KUKA KRL program: Milling_2_2.src

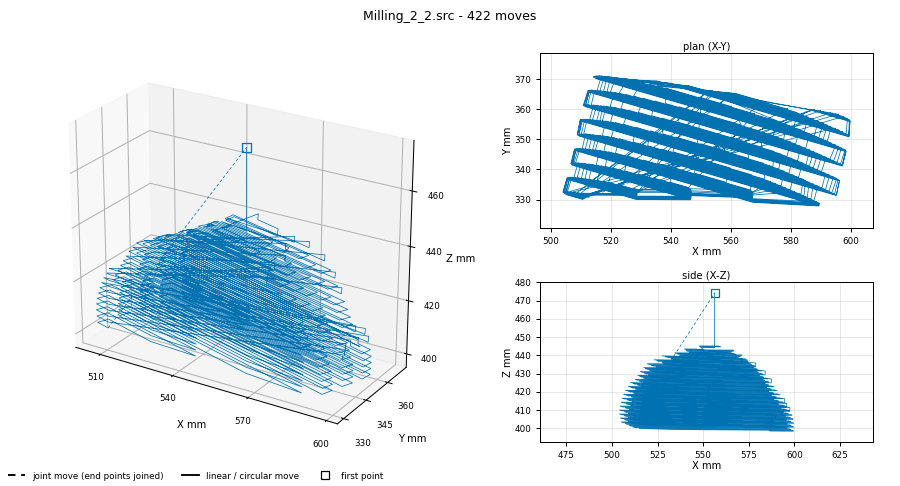
[picture p0: tool path of Milling_2_2.src, 422 of 424 moves have a stored position in this frame; points joined in program order, loops and branches not executed]
&ACCESS RVP
&REL 1
&PARAM TEMPLATE = C:\KRC\Roboter\Template\vorgabe
&PARAM EDITMASK = *
DEF Milling_2_2 ( )


;FOLD INI
;FOLD BASISTECH INI
GLOBAL INTERRUPT DECL 3 WHEN $STOPMESS==TRUE DO IR_STOPM ( )
INTERRUPT ON 3
BAS (#INITMOV,0 )
;ENDFOLD (BASISTECH INI)
;ENDFOLD (INI)

;FOLD STARTPOSITION - BASE IS 0, TOOL IS 5, SPEED IS 15%, POSITION IS A1 5,A2 -90,A3 100,A4 5,A5 -10,A6 -5,E1 0,E2 0,E3 0,E4 0
$BWDSTART = FALSE
PDAT_ACT = {VEL 15,ACC 100,APO_DIST 50}
FDAT_ACT = {TOOL_NO 5,BASE_NO 0,IPO_FRAME #BASE}
BAS (#PTP_PARAMS,15)
PTP  {A1 5,A2 -90,A3 100,A4 5,A5 -10,A6 -5,E1 0,E2 0,E3 0,E4 0}
;ENDFOLD

;FOLD LIN SPEED IS 0.1 m/sec, INTERPOLATION SETTINGS IN FOLD
$VEL.CP=0.1
$ADVANCE=3
;ENDFOLD

BAS(#VEL_PTP,2)
PTP {X 556.311, Y 346.712, Z 474.273, A -110.612, B 84.801, C -94.37, E1 0, E2 0, E3 0, E4 0, S 'B010'}
$VEL.CP=0.012
LIN {X 556.311, Y 346.712, Z 444.273, A -110.612, B 84.801, C -94.37, E1 0, E2 0, E3 0, E4 0}
LIN {X 549.895, Y 348.583, Z 444.319, A -110.612, B 84.801, C -94.37, E1 0, E2 0, E3 0, E4 0}
LIN {X 548.876, Y 343.693, Z 444.768, A -110.612, B 84.801, C -94.37, E1 0, E2 0, E3 0, E4 0}
LIN {X 559.743, Y 340.524, Z 444.69, A -110.612, B 84.801, C -94.37, E1 0, E2 0, E3 0, E4 0}
LIN {X 558.354, Y 335.742, Z 445.142, A -110.612, B 84.801, C -94.37, E1 0, E2 0, E3 0, E4 0}
LIN {X 547.877, Y 338.798, Z 445.217, A -110.612, B 84.801, C -94.37, E1 0, E2 0, E3 0, E4 0}
LIN {X 550.299, Y 364.027, Z 442.992, A -110.612, B 84.801, C -94.37, E1 0, E2 0, E3 0, E4 0}
LIN {X 550.229, Y 363.842, Z 440.827, A -110.612, B 84.801, C -94.37, E1 0, E2 0, E3 0, E4 0}
LIN {X 560.058, Y 360.976, Z 440.756, A -110.612, B 84.801, C -94.37, E1 0, E2 0, E3 0, E4 0}
LIN {X 563.393, Y 354.816, Z 441.174, A -110.612, B 84.801, C -94.37, E1 0, E2 0, E3 0, E4 0}
LIN {X 542.631, Y 360.871, Z 441.323, A -110.612, B 84.801, C -94.37, E1 0, E2 0, E3 0, E4 0}
LIN {X 542.344, Y 355.768, Z 441.767, A -110.612, B 84.801, C -94.37, E1 0, E2 0, E3 0, E4 0}
LIN {X 565.078, Y 349.137, Z 441.603, A -110.612, B 84.801, C -94.37, E1 0, E2 0, E3 0, E4 0}
LIN {X 565.885, Y 343.715, Z 442.039, A -110.612, B 84.801, C -94.37, E1 0, E2 0, E3 0, E4 0}
LIN {X 541.583, Y 350.803, Z 442.214, A -110.612, B 84.801, C -94.37, E1 0, E2 0, E3 0, E4 0}
LIN {X 540.685, Y 345.878, Z 442.662, A -110.612, B 84.801, C -94.37, E1 0, E2 0, E3 0, E4 0}
LIN {X 566.796, Y 338.262, Z 442.474, A -110.612, B 84.801, C -94.37, E1 0, E2 0, E3 0, E4 0}
LIN {X 566.499, Y 333.162, Z 442.918, A -110.612, B 84.801, C -94.37, E1 0, E2 0, E3 0, E4 0}
LIN {X 540.83, Y 340.648, Z 443.103, A -110.612, B 84.801, C -94.37, E1 0, E2 0, E3 0, E4 0}
LIN {X 539.697, Y 335.792, Z 443.553, A -110.612, B 84.801, C -94.37, E1 0, E2 0, E3 0, E4 0}
LIN {X 545.888, Y 333.986, Z 443.508, A -110.612, B 84.801, C -94.37, E1 0, E2 0, E3 0, E4 0}
LIN {X 567.928, Y 358.68, Z 440.699, A -110.612, B 84.801, C -94.37, E1 0, E2 0, E3 0, E4 0}
LIN {X 567.859, Y 358.496, Z 438.534, A -110.612, B 84.801, C -94.37, E1 0, E2 0, E3 0, E4 0}
LIN {X 538.218, Y 367.141, Z 438.747, A -110.612, B 84.801, C -94.37, E1 0, E2 0, E3 0, E4 0}
LIN {X 538.244, Y 361.946, Z 439.189, A -110.612, B 84.801, C -94.37, E1 0, E2 0, E3 0, E4 0}
LIN {X 569.164, Y 352.928, Z 438.966, A -110.612, B 84.801, C -94.37, E1 0, E2 0, E3 0, E4 0}
LIN {X 570.368, Y 347.39, Z 439.399, A -110.612, B 84.801, C -94.37, E1 0, E2 0, E3 0, E4 0}
LIN {X 536.951, Y 357.136, Z 439.64, A -110.612, B 84.801, C -94.37, E1 0, E2 0, E3 0, E4 0}
LIN {X 537.304, Y 351.846, Z 440.079, A -110.612, B 84.801, C -94.37, E1 0, E2 0, E3 0, E4 0}
LIN {X 570.875, Y 342.055, Z 439.837, A -110.612, B 84.801, C -94.37, E1 0, E2 0, E3 0, E4 0}
LIN {X 571.155, Y 336.786, Z 440.277, A -110.612, B 84.801, C -94.37, E1 0, E2 0, E3 0, E4 0}
LIN {X 536.952, Y 346.762, Z 440.523, A -110.612, B 84.801, C -94.37, E1 0, E2 0, E3 0, E4 0}
LIN {X 535.523, Y 341.992, Z 440.975, A -110.612, B 84.801, C -94.37, E1 0, E2 0, E3 0, E4 0}
LIN {X 566.961, Y 332.823, Z 440.749, A -110.612, B 84.801, C -94.37, E1 0, E2 0, E3 0, E4 0}
LIN {X 546.398, Y 333.633, Z 441.339, A -110.612, B 84.801, C -94.37, E1 0, E2 0, E3 0, E4 0}
LIN {X 534.432, Y 337.123, Z 441.425, A -110.612, B 84.801, C -94.37, E1 0, E2 0, E3 0, E4 0}
LIN {X 571.445, Y 362.637, Z 438.067, A -110.612, B 84.801, C -94.37, E1 0, E2 0, E3 0, E4 0}
LIN {X 571.376, Y 362.452, Z 435.902, A -110.612, B 84.801, C -94.37, E1 0, E2 0, E3 0, E4 0}
LIN {X 561.675, Y 365.282, Z 435.971, A -110.612, B 84.801, C -94.37, E1 0, E2 0, E3 0, E4 0}
LIN {X 535.453, Y 367.743, Z 436.602, A -110.612, B 84.801, C -94.37, E1 0, E2 0, E3 0, E4 0}
LIN {X 574.931, Y 356.229, Z 436.318, A -110.612, B 84.801, C -94.37, E1 0, E2 0, E3 0, E4 0}
LIN {X 574.139, Y 351.273, Z 436.765, A -110.612, B 84.801, C -94.37, E1 0, E2 0, E3 0, E4 0}
LIN {X 534.55, Y 362.819, Z 437.05, A -110.612, B 84.801, C -94.37, E1 0, E2 0, E3 0, E4 0}
LIN {X 533.571, Y 357.917, Z 437.499, A -110.612, B 84.801, C -94.37, E1 0, E2 0, E3 0, E4 0}
LIN {X 574.308, Y 346.036, Z 437.206, A -110.612, B 84.801, C -94.37, E1 0, E2 0, E3 0, E4 0}
LIN {X 573.943, Y 340.956, Z 437.65, A -110.612, B 84.801, C -94.37, E1 0, E2 0, E3 0, E4 0}
LIN {X 533.122, Y 352.862, Z 437.944, A -110.612, B 84.801, C -94.37, E1 0, E2 0, E3 0, E4 0}
LIN {X 532.259, Y 347.926, Z 438.392, A -110.612, B 84.801, C -94.37, E1 0, E2 0, E3 0, E4 0}
LIN {X 573.267, Y 335.966, Z 438.097, A -110.612, B 84.801, C -94.37, E1 0, E2 0, E3 0, E4 0}
LIN {X 567.221, Y 332.542, Z 438.582, A -110.612, B 84.801, C -94.37, E1 0, E2 0, E3 0, E4 0}
LIN {X 530.884, Y 343.14, Z 438.843, A -110.612, B 84.801, C -94.37, E1 0, E2 0, E3 0, E4 0}
LIN {X 529.176, Y 338.451, Z 439.297, A -110.612, B 84.801, C -94.37, E1 0, E2 0, E3 0, E4 0}
LIN {X 546.678, Y 333.347, Z 439.171, A -110.612, B 84.801, C -94.37, E1 0, E2 0, E3 0, E4 0}
LIN {X 528.874, Y 333.353, Z 439.741, A -110.612, B 84.801, C -94.37, E1 0, E2 0, E3 0, E4 0}
LIN {X 527.487, Y 333.757, Z 439.751, A -110.612, B 84.801, C -94.37, E1 0, E2 0, E3 0, E4 0}
LIN {X 578.837, Y 360.276, Z 435.848, A -110.612, B 84.801, C -94.37, E1 0, E2 0, E3 0, E4 0}
LIN {X 578.768, Y 360.092, Z 433.683, A -110.612, B 84.801, C -94.37, E1 0, E2 0, E3 0, E4 0}
LIN {X 561.03, Y 365.265, Z 433.811, A -110.612, B 84.801, C -94.37, E1 0, E2 0, E3 0, E4 0}
LIN {X 532.693, Y 368.343, Z 434.456, A -110.612, B 84.801, C -94.37, E1 0, E2 0, E3 0, E4 0}
LIN {X 578.339, Y 355.03, Z 434.128, A -110.612, B 84.801, C -94.37, E1 0, E2 0, E3 0, E4 0}
LIN {X 577.543, Y 350.075, Z 434.575, A -110.612, B 84.801, C -94.37, E1 0, E2 0, E3 0, E4 0}
LIN {X 530.911, Y 363.676, Z 434.911, A -110.612, B 84.801, C -94.37, E1 0, E2 0, E3 0, E4 0}
LIN {X 529.165, Y 358.998, Z 435.365, A -110.612, B 84.801, C -94.37, E1 0, E2 0, E3 0, E4 0}
LIN {X 576.615, Y 345.159, Z 435.023, A -110.612, B 84.801, C -94.37, E1 0, E2 0, E3 0, E4 0}
LIN {X 575.918, Y 340.175, Z 435.47, A -110.612, B 84.801, C -94.37, E1 0, E2 0, E3 0, E4 0}
LIN {X 528.335, Y 354.053, Z 435.813, A -110.612, B 84.801, C -94.37, E1 0, E2 0, E3 0, E4 0}
LIN {X 527.42, Y 349.133, Z 436.261, A -110.612, B 84.801, C -94.37, E1 0, E2 0, E3 0, E4 0}
LIN {X 574.963, Y 335.266, Z 435.919, A -110.612, B 84.801, C -94.37, E1 0, E2 0, E3 0, E4 0}
LIN {X 567.23, Y 332.335, Z 436.416, A -110.612, B 84.801, C -94.37, E1 0, E2 0, E3 0, E4 0}
LIN {X 525.837, Y 344.408, Z 436.714, A -110.612, B 84.801, C -94.37, E1 0, E2 0, E3 0, E4 0}
LIN {X 524.56, Y 339.593, Z 437.165, A -110.612, B 84.801, C -94.37, E1 0, E2 0, E3 0, E4 0}
LIN {X 546.693, Y 333.138, Z 437.006, A -110.612, B 84.801, C -94.37, E1 0, E2 0, E3 0, E4 0}
LIN {X 528.865, Y 333.151, Z 437.576, A -110.612, B 84.801, C -94.37, E1 0, E2 0, E3 0, E4 0}
LIN {X 523.143, Y 334.819, Z 437.617, A -110.612, B 84.801, C -94.37, E1 0, E2 0, E3 0, E4 0}
LIN {X 560.537, Y 365.409, Z 433.814, A -110.612, B 84.801, C -94.37, E1 0, E2 0, E3 0, E4 0}
LIN {X 560.468, Y 365.225, Z 431.649, A -110.612, B 84.801, C -94.37, E1 0, E2 0, E3 0, E4 0}
LIN {X 581.97, Y 358.954, Z 431.495, A -110.612, B 84.801, C -94.37, E1 0, E2 0, E3 0, E4 0}
LIN {X 580.949, Y 354.064, Z 431.944, A -110.612, B 84.801, C -94.37, E1 0, E2 0, E3 0, E4 0}
LIN {X 530.225, Y 368.858, Z 432.308, A -110.612, B 84.801, C -94.37, E1 0, E2 0, E3 0, E4 0}
LIN {X 527.54, Y 364.454, Z 432.769, A -110.612, B 84.801, C -94.37, E1 0, E2 0, E3 0, E4 0}
LIN {X 579.85, Y 349.198, Z 432.393, A -110.612, B 84.801, C -94.37, E1 0, E2 0, E3 0, E4 0}
LIN {X 578.612, Y 344.372, Z 432.844, A -110.612, B 84.801, C -94.37, E1 0, E2 0, E3 0, E4 0}
LIN {X 525.917, Y 359.741, Z 433.223, A -110.612, B 84.801, C -94.37, E1 0, E2 0, E3 0, E4 0}
LIN {X 524.197, Y 355.055, Z 433.677, A -110.612, B 84.801, C -94.37, E1 0, E2 0, E3 0, E4 0}
LIN {X 577.658, Y 339.463, Z 433.292, A -110.612, B 84.801, C -94.37, E1 0, E2 0, E3 0, E4 0}
LIN {X 576.646, Y 334.571, Z 433.741, A -110.612, B 84.801, C -94.37, E1 0, E2 0, E3 0, E4 0}
LIN {X 522.84, Y 350.264, Z 434.128, A -110.612, B 84.801, C -94.37, E1 0, E2 0, E3 0, E4 0}
LIN {X 521.544, Y 345.455, Z 434.58, A -110.612, B 84.801, C -94.37, E1 0, E2 0, E3 0, E4 0}
LIN {X 567.264, Y 332.12, Z 434.251, A -110.612, B 84.801, C -94.37, E1 0, E2 0, E3 0, E4 0}
LIN {X 546.731, Y 332.922, Z 434.84, A -110.612, B 84.801, C -94.37, E1 0, E2 0, E3 0, E4 0}
LIN {X 520.683, Y 340.519, Z 435.027, A -110.612, B 84.801, C -94.37, E1 0, E2 0, E3 0, E4 0}
LIN {X 519.275, Y 335.743, Z 435.479, A -110.612, B 84.801, C -94.37, E1 0, E2 0, E3 0, E4 0}
LIN {X 528.883, Y 332.941, Z 435.41, A -110.612, B 84.801, C -94.37, E1 0, E2 0, E3 0, E4 0}
LIN {X 584.039, Y 358.35, Z 431.48, A -110.612, B 84.801, C -94.37, E1 0, E2 0, E3 0, E4 0}
LIN {X 583.969, Y 358.166, Z 429.315, A -110.612, B 84.801, C -94.37, E1 0, E2 0, E3 0, E4 0}
LIN {X 560.841, Y 364.911, Z 429.481, A -110.612, B 84.801, C -94.37, E1 0, E2 0, E3 0, E4 0}
LIN {X 527.741, Y 369.378, Z 430.161, A -110.612, B 84.801, C -94.37, E1 0, E2 0, E3 0, E4 0}
LIN {X 582.834, Y 353.31, Z 429.765, A -110.612, B 84.801, C -94.37, E1 0, E2 0, E3 0, E4 0}
LIN {X 581.5, Y 348.512, Z 430.216, A -110.612, B 84.801, C -94.37, E1 0, E2 0, E3 0, E4 0}
LIN {X 525.057, Y 364.974, Z 430.622, A -110.612, B 84.801, C -94.37, E1 0, E2 0, E3 0, E4 0}
LIN {X 523.33, Y 360.291, Z 431.076, A -110.612, B 84.801, C -94.37, E1 0, E2 0, E3 0, E4 0}
LIN {X 580.316, Y 343.67, Z 430.666, A -110.612, B 84.801, C -94.37, E1 0, E2 0, E3 0, E4 0}
LIN {X 579.317, Y 338.775, Z 431.115, A -110.612, B 84.801, C -94.37, E1 0, E2 0, E3 0, E4 0}
LIN {X 521.512, Y 355.634, Z 431.531, A -110.612, B 84.801, C -94.37, E1 0, E2 0, E3 0, E4 0}
LIN {X 520.22, Y 350.824, Z 431.982, A -110.612, B 84.801, C -94.37, E1 0, E2 0, E3 0, E4 0}
LIN {X 578.198, Y 333.914, Z 431.565, A -110.612, B 84.801, C -94.37, E1 0, E2 0, E3 0, E4 0}
LIN {X 567.291, Y 331.908, Z 432.085, A -110.612, B 84.801, C -94.37, E1 0, E2 0, E3 0, E4 0}
LIN {X 519.262, Y 345.916, Z 432.43, A -110.612, B 84.801, C -94.37, E1 0, E2 0, E3 0, E4 0}
LIN {X 518.103, Y 341.067, Z 432.88, A -110.612, B 84.801, C -94.37, E1 0, E2 0, E3 0, E4 0}
LIN {X 546.763, Y 332.708, Z 432.674, A -110.612, B 84.801, C -94.37, E1 0, E2 0, E3 0, E4 0}
LIN {X 528.89, Y 332.734, Z 433.244, A -110.612, B 84.801, C -94.37, E1 0, E2 0, E3 0, E4 0}
LIN {X 517.363, Y 336.096, Z 433.327, A -110.612, B 84.801, C -94.37, E1 0, E2 0, E3 0, E4 0}
LIN {X 560.576, Y 364.988, Z 429.483, A -110.612, B 84.801, C -94.37, E1 0, E2 0, E3 0, E4 0}
LIN {X 560.507, Y 364.804, Z 427.318, A -110.612, B 84.801, C -94.37, E1 0, E2 0, E3 0, E4 0}
LIN {X 585.6, Y 357.486, Z 427.137, A -110.612, B 84.801, C -94.37, E1 0, E2 0, E3 0, E4 0}
LIN {X 584.414, Y 352.645, Z 427.587, A -110.612, B 84.801, C -94.37, E1 0, E2 0, E3 0, E4 0}
LIN {X 525.529, Y 369.819, Z 428.011, A -110.612, B 84.801, C -94.37, E1 0, E2 0, E3 0, E4 0}
LIN {X 522.763, Y 365.439, Z 428.473, A -110.612, B 84.801, C -94.37, E1 0, E2 0, E3 0, E4 0}
LIN {X 583.251, Y 347.796, Z 428.038, A -110.612, B 84.801, C -94.37, E1 0, E2 0, E3 0, E4 0}
LIN {X 582.149, Y 342.931, Z 428.487, A -110.612, B 84.801, C -94.37, E1 0, E2 0, E3 0, E4 0}
LIN {X 521.328, Y 360.67, Z 428.925, A -110.612, B 84.801, C -94.37, E1 0, E2 0, E3 0, E4 0}
LIN {X 519.9, Y 355.9, Z 429.377, A -110.612, B 84.801, C -94.37, E1 0, E2 0, E3 0, E4 0}
LIN {X 580.925, Y 338.101, Z 428.938, A -110.612, B 84.801, C -94.37, E1 0, E2 0, E3 0, E4 0}
LIN {X 579.682, Y 333.276, Z 429.389, A -110.612, B 84.801, C -94.37, E1 0, E2 0, E3 0, E4 0}
LIN {X 518.74, Y 351.051, Z 429.827, A -110.612, B 84.801, C -94.37, E1 0, E2 0, E3 0, E4 0}
LIN {X 517.721, Y 346.161, Z 430.276, A -110.612, B 84.801, C -94.37, E1 0, E2 0, E3 0, E4 0}
LIN {X 567.295, Y 331.702, Z 429.919, A -110.612, B 84.801, C -94.37, E1 0, E2 0, E3 0, E4 0}
LIN {X 546.773, Y 332.5, Z 430.509, A -110.612, B 84.801, C -94.37, E1 0, E2 0, E3 0, E4 0}
LIN {X 516.775, Y 341.25, Z 430.724, A -110.612, B 84.801, C -94.37, E1 0, E2 0, E3 0, E4 0}
LIN {X 515.501, Y 336.434, Z 431.175, A -110.612, B 84.801, C -94.37, E1 0, E2 0, E3 0, E4 0}
LIN {X 528.872, Y 332.535, Z 431.079, A -110.612, B 84.801, C -94.37, E1 0, E2 0, E3 0, E4 0}
LIN {X 587.401, Y 356.96, Z 427.124, A -110.612, B 84.801, C -94.37, E1 0, E2 0, E3 0, E4 0}
LIN {X 587.331, Y 356.776, Z 424.959, A -110.612, B 84.801, C -94.37, E1 0, E2 0, E3 0, E4 0}
LIN {X 558.579, Y 365.162, Z 425.166, A -110.612, B 84.801, C -94.37, E1 0, E2 0, E3 0, E4 0}
LIN {X 523.134, Y 370.313, Z 425.863, A -110.612, B 84.801, C -94.37, E1 0, E2 0, E3 0, E4 0}
LIN {X 586.126, Y 351.94, Z 425.41, A -110.612, B 84.801, C -94.37, E1 0, E2 0, E3 0, E4 0}
LIN {X 584.86, Y 347.123, Z 425.861, A -110.612, B 84.801, C -94.37, E1 0, E2 0, E3 0, E4 0}
LIN {X 521.221, Y 365.684, Z 426.318, A -110.612, B 84.801, C -94.37, E1 0, E2 0, E3 0, E4 0}
LIN {X 519.757, Y 360.924, Z 426.771, A -110.612, B 84.801, C -94.37, E1 0, E2 0, E3 0, E4 0}
LIN {X 583.82, Y 342.239, Z 426.31, A -110.612, B 84.801, C -94.37, E1 0, E2 0, E3 0, E4 0}
LIN {X 582.502, Y 337.436, Z 426.761, A -110.612, B 84.801, C -94.37, E1 0, E2 0, E3 0, E4 0}
LIN {X 518.3, Y 356.162, Z 427.223, A -110.612, B 84.801, C -94.37, E1 0, E2 0, E3 0, E4 0}
LIN {X 517.173, Y 351.303, Z 427.673, A -110.612, B 84.801, C -94.37, E1 0, E2 0, E3 0, E4 0}
LIN {X 581.23, Y 332.62, Z 427.212, A -110.612, B 84.801, C -94.37, E1 0, E2 0, E3 0, E4 0}
LIN {X 567.31, Y 331.493, Z 427.754, A -110.612, B 84.801, C -94.37, E1 0, E2 0, E3 0, E4 0}
LIN {X 516.211, Y 346.397, Z 428.121, A -110.612, B 84.801, C -94.37, E1 0, E2 0, E3 0, E4 0}
LIN {X 515.15, Y 341.519, Z 428.571, A -110.612, B 84.801, C -94.37, E1 0, E2 0, E3 0, E4 0}
LIN {X 546.795, Y 332.289, Z 428.343, A -110.612, B 84.801, C -94.37, E1 0, E2 0, E3 0, E4 0}
LIN {X 528.864, Y 332.332, Z 428.914, A -110.612, B 84.801, C -94.37, E1 0, E2 0, E3 0, E4 0}
LIN {X 514.073, Y 336.646, Z 429.02, A -110.612, B 84.801, C -94.37, E1 0, E2 0, E3 0, E4 0}
LIN {X 555.834, Y 365.962, Z 425.186, A -110.612, B 84.801, C -94.37, E1 0, E2 0, E3 0, E4 0}
LIN {X 555.764, Y 365.778, Z 423.021, A -110.612, B 84.801, C -94.37, E1 0, E2 0, E3 0, E4 0}
LIN {X 589.011, Y 356.081, Z 422.782, A -110.612, B 84.801, C -94.37, E1 0, E2 0, E3 0, E4 0}
LIN {X 587.7, Y 351.277, Z 423.233, A -110.612, B 84.801, C -94.37, E1 0, E2 0, E3 0, E4 0}
LIN {X 521.625, Y 370.548, Z 423.708, A -110.612, B 84.801, C -94.37, E1 0, E2 0, E3 0, E4 0}
LIN {X 519.881, Y 365.87, Z 424.163, A -110.612, B 84.801, C -94.37, E1 0, E2 0, E3 0, E4 0}
LIN {X 586.204, Y 346.526, Z 423.686, A -110.612, B 84.801, C -94.37, E1 0, E2 0, E3 0, E4 0}
LIN {X 584.986, Y 341.694, Z 424.136, A -110.612, B 84.801, C -94.37, E1 0, E2 0, E3 0, E4 0}
LIN {X 518.482, Y 361.091, Z 424.614, A -110.612, B 84.801, C -94.37, E1 0, E2 0, E3 0, E4 0}
LIN {X 517.199, Y 356.278, Z 425.065, A -110.612, B 84.801, C -94.37, E1 0, E2 0, E3 0, E4 0}
LIN {X 584.056, Y 336.779, Z 424.584, A -110.612, B 84.801, C -94.37, E1 0, E2 0, E3 0, E4 0}
LIN {X 583.256, Y 331.825, Z 425.032, A -110.612, B 84.801, C -94.37, E1 0, E2 0, E3 0, E4 0}
LIN {X 516.269, Y 351.362, Z 425.514, A -110.612, B 84.801, C -94.37, E1 0, E2 0, E3 0, E4 0}
LIN {X 514.87, Y 346.583, Z 425.965, A -110.612, B 84.801, C -94.37, E1 0, E2 0, E3 0, E4 0}
LIN {X 567.242, Y 331.309, Z 425.589, A -110.612, B 84.801, C -94.37, E1 0, E2 0, E3 0, E4 0}
LIN {X 546.728, Y 332.105, Z 426.178, A -110.612, B 84.801, C -94.37, E1 0, E2 0, E3 0, E4 0}
LIN {X 513.756, Y 341.721, Z 426.415, A -110.612, B 84.801, C -94.37, E1 0, E2 0, E3 0, E4 0}
LIN {X 512.754, Y 336.826, Z 426.864, A -110.612, B 84.801, C -94.37, E1 0, E2 0, E3 0, E4 0}
LIN {X 528.791, Y 332.149, Z 426.749, A -110.612, B 84.801, C -94.37, E1 0, E2 0, E3 0, E4 0}
LIN {X 553.831, Y 366.342, Z 423.035, A -110.612, B 84.801, C -94.37, E1 0, E2 0, E3 0, E4 0}
LIN {X 553.761, Y 366.158, Z 420.87, A -110.612, B 84.801, C -94.37, E1 0, E2 0, E3 0, E4 0}
LIN {X 590.695, Y 355.386, Z 420.604, A -110.612, B 84.801, C -94.37, E1 0, E2 0, E3 0, E4 0}
LIN {X 589.228, Y 350.627, Z 421.056, A -110.612, B 84.801, C -94.37, E1 0, E2 0, E3 0, E4 0}
LIN {X 520.009, Y 370.815, Z 421.554, A -110.612, B 84.801, C -94.37, E1 0, E2 0, E3 0, E4 0}
LIN {X 518.731, Y 366.001, Z 422.005, A -110.612, B 84.801, C -94.37, E1 0, E2 0, E3 0, E4 0}
LIN {X 587.548, Y 345.93, Z 421.51, A -110.612, B 84.801, C -94.37, E1 0, E2 0, E3 0, E4 0}
LIN {X 586.024, Y 341.187, Z 421.963, A -110.612, B 84.801, C -94.37, E1 0, E2 0, E3 0, E4 0}
LIN {X 517.512, Y 361.169, Z 422.456, A -110.612, B 84.801, C -94.37, E1 0, E2 0, E3 0, E4 0}
LIN {X 516.338, Y 356.324, Z 422.906, A -110.612, B 84.801, C -94.37, E1 0, E2 0, E3 0, E4 0}
LIN {X 584.869, Y 336.337, Z 422.413, A -110.612, B 84.801, C -94.37, E1 0, E2 0, E3 0, E4 0}
LIN {X 584.263, Y 331.326, Z 422.859, A -110.612, B 84.801, C -94.37, E1 0, E2 0, E3 0, E4 0}
LIN {X 515.26, Y 351.452, Z 423.355, A -110.612, B 84.801, C -94.37, E1 0, E2 0, E3 0, E4 0}
LIN {X 513.944, Y 346.649, Z 423.806, A -110.612, B 84.801, C -94.37, E1 0, E2 0, E3 0, E4 0}
LIN {X 567.24, Y 331.104, Z 423.423, A -110.612, B 84.801, C -94.37, E1 0, E2 0, E3 0, E4 0}
LIN {X 546.734, Y 331.898, Z 424.013, A -110.612, B 84.801, C -94.37, E1 0, E2 0, E3 0, E4 0}
LIN {X 512.57, Y 341.862, Z 424.258, A -110.612, B 84.801, C -94.37, E1 0, E2 0, E3 0, E4 0}
LIN {X 511.41, Y 337.014, Z 424.708, A -110.612, B 84.801, C -94.37, E1 0, E2 0, E3 0, E4 0}
LIN {X 528.764, Y 331.952, Z 424.583, A -110.612, B 84.801, C -94.37, E1 0, E2 0, E3 0, E4 0}
LIN {X 510.469, Y 332.101, Z 425.157, A -110.612, B 84.801, C -94.37, E1 0, E2 0, E3 0, E4 0}
LIN {X 510.134, Y 332.199, Z 425.159, A -110.612, B 84.801, C -94.37, E1 0, E2 0, E3 0, E4 0}
LIN {X 552.927, Y 366.401, Z 420.876, A -110.612, B 84.801, C -94.37, E1 0, E2 0, E3 0, E4 0}
LIN {X 552.857, Y 366.217, Z 418.711, A -110.612, B 84.801, C -94.37, E1 0, E2 0, E3 0, E4 0}
LIN {X 592.136, Y 354.761, Z 418.428, A -110.612, B 84.801, C -94.37, E1 0, E2 0, E3 0, E4 0}
LIN {X 590.642, Y 350.009, Z 418.881, A -110.612, B 84.801, C -94.37, E1 0, E2 0, E3 0, E4 0}
LIN {X 518.742, Y 370.98, Z 419.398, A -110.612, B 84.801, C -94.37, E1 0, E2 0, E3 0, E4 0}
LIN {X 517.598, Y 366.127, Z 419.848, A -110.612, B 84.801, C -94.37, E1 0, E2 0, E3 0, E4 0}
LIN {X 588.889, Y 345.334, Z 419.335, A -110.612, B 84.801, C -94.37, E1 0, E2 0, E3 0, E4 0}
LIN {X 587.367, Y 340.591, Z 419.788, A -110.612, B 84.801, C -94.37, E1 0, E2 0, E3 0, E4 0}
LIN {X 516.578, Y 361.237, Z 420.297, A -110.612, B 84.801, C -94.37, E1 0, E2 0, E3 0, E4 0}
LIN {X 515.325, Y 356.415, Z 420.748, A -110.612, B 84.801, C -94.37, E1 0, E2 0, E3 0, E4 0}
LIN {X 586.011, Y 335.799, Z 420.239, A -110.612, B 84.801, C -94.37, E1 0, E2 0, E3 0, E4 0}
LIN {X 585.368, Y 330.8, Z 420.686, A -110.612, B 84.801, C -94.37, E1 0, E2 0, E3 0, E4 0}
LIN {X 513.956, Y 351.628, Z 421.199, A -110.612, B 84.801, C -94.37, E1 0, E2 0, E3 0, E4 0}
LIN {X 512.647, Y 346.822, Z 421.651, A -110.612, B 84.801, C -94.37, E1 0, E2 0, E3 0, E4 0}
LIN {X 567.238, Y 330.9, Z 421.258, A -110.612, B 84.801, C -94.37, E1 0, E2 0, E3 0, E4 0}
LIN {X 546.738, Y 331.693, Z 421.847, A -110.612, B 84.801, C -94.37, E1 0, E2 0, E3 0, E4 0}
LIN {X 511.345, Y 342.015, Z 422.102, A -110.612, B 84.801, C -94.37, E1 0, E2 0, E3 0, E4 0}
LIN {X 510.226, Y 337.154, Z 422.551, A -110.612, B 84.801, C -94.37, E1 0, E2 0, E3 0, E4 0}
LIN {X 528.74, Y 331.755, Z 422.418, A -110.612, B 84.801, C -94.37, E1 0, E2 0, E3 0, E4 0}
LIN {X 510.485, Y 331.892, Z 422.991, A -110.612, B 84.801, C -94.37, E1 0, E2 0, E3 0, E4 0}
LIN {X 508.837, Y 332.373, Z 423.003, A -110.612, B 84.801, C -94.37, E1 0, E2 0, E3 0, E4 0}
LIN {X 552.608, Y 366.29, Z 418.713, A -110.612, B 84.801, C -94.37, E1 0, E2 0, E3 0, E4 0}
LIN {X 552.539, Y 366.105, Z 416.548, A -110.612, B 84.801, C -94.37, E1 0, E2 0, E3 0, E4 0}
LIN {X 593.359, Y 354.2, Z 416.254, A -110.612, B 84.801, C -94.37, E1 0, E2 0, E3 0, E4 0}
LIN {X 592.023, Y 349.402, Z 416.706, A -110.612, B 84.801, C -94.37, E1 0, E2 0, E3 0, E4 0}
LIN {X 517.881, Y 371.027, Z 417.239, A -110.612, B 84.801, C -94.37, E1 0, E2 0, E3 0, E4 0}
LIN {X 516.358, Y 366.284, Z 417.691, A -110.612, B 84.801, C -94.37, E1 0, E2 0, E3 0, E4 0}
LIN {X 590.217, Y 344.742, Z 417.16, A -110.612, B 84.801, C -94.37, E1 0, E2 0, E3 0, E4 0}
LIN {X 588.756, Y 339.981, Z 417.612, A -110.612, B 84.801, C -94.37, E1 0, E2 0, E3 0, E4 0}
LIN {X 515.373, Y 361.384, Z 418.14, A -110.612, B 84.801, C -94.37, E1 0, E2 0, E3 0, E4 0}
LIN {X 513.91, Y 356.624, Z 418.592, A -110.612, B 84.801, C -94.37, E1 0, E2 0, E3 0, E4 0}
LIN {X 587.433, Y 335.18, Z 418.064, A -110.612, B 84.801, C -94.37, E1 0, E2 0, E3 0, E4 0}
LIN {X 586.59, Y 330.239, Z 418.512, A -110.612, B 84.801, C -94.37, E1 0, E2 0, E3 0, E4 0}
LIN {X 512.808, Y 351.758, Z 419.042, A -110.612, B 84.801, C -94.37, E1 0, E2 0, E3 0, E4 0}
LIN {X 511.535, Y 346.942, Z 419.493, A -110.612, B 84.801, C -94.37, E1 0, E2 0, E3 0, E4 0}
LIN {X 567.23, Y 330.698, Z 419.093, A -110.612, B 84.801, C -94.37, E1 0, E2 0, E3 0, E4 0}
LIN {X 546.736, Y 331.489, Z 419.682, A -110.612, B 84.801, C -94.37, E1 0, E2 0, E3 0, E4 0}
LIN {X 510.218, Y 342.139, Z 419.944, A -110.612, B 84.801, C -94.37, E1 0, E2 0, E3 0, E4 0}
LIN {X 508.801, Y 337.365, Z 420.396, A -110.612, B 84.801, C -94.37, E1 0, E2 0, E3 0, E4 0}
LIN {X 528.709, Y 331.559, Z 420.253, A -110.612, B 84.801, C -94.37, E1 0, E2 0, E3 0, E4 0}
LIN {X 510.496, Y 331.684, Z 420.826, A -110.612, B 84.801, C -94.37, E1 0, E2 0, E3 0, E4 0}
LIN {X 507.498, Y 332.558, Z 420.847, A -110.612, B 84.801, C -94.37, E1 0, E2 0, E3 0, E4 0}
LIN {X 594.753, Y 353.793, Z 416.244, A -110.612, B 84.801, C -94.37, E1 0, E2 0, E3 0, E4 0}
LIN {X 594.684, Y 353.609, Z 414.079, A -110.612, B 84.801, C -94.37, E1 0, E2 0, E3 0, E4 0}
LIN {X 553.923, Y 365.497, Z 414.372, A -110.612, B 84.801, C -94.37, E1 0, E2 0, E3 0, E4 0}
LIN {X 545.227, Y 368.033, Z 414.435, A -110.612, B 84.801, C -94.37, E1 0, E2 0, E3 0, E4 0}
LIN {X 549.101, Y 366.903, Z 414.407, A -110.612, B 84.801, C -94.37, E1 0, E2 0, E3 0, E4 0}
LIN {X 593.422, Y 348.79, Z 414.53, A -110.612, B 84.801, C -94.37, E1 0, E2 0, E3 0, E4 0}
LIN {X 516.863, Y 371.119, Z 415.08, A -110.612, B 84.801, C -94.37, E1 0, E2 0, E3 0, E4 0}
LIN {X 515.434, Y 366.349, Z 415.532, A -110.612, B 84.801, C -94.37, E1 0, E2 0, E3 0, E4 0}
LIN {X 591.641, Y 344.122, Z 414.984, A -110.612, B 84.801, C -94.37, E1 0, E2 0, E3 0, E4 0}
LIN {X 590.145, Y 339.371, Z 415.437, A -110.612, B 84.801, C -94.37, E1 0, E2 0, E3 0, E4 0}
LIN {X 514.282, Y 361.497, Z 415.982, A -110.612, B 84.801, C -94.37, E1 0, E2 0, E3 0, E4 0}
LIN {X 512.939, Y 356.702, Z 416.434, A -110.612, B 84.801, C -94.37, E1 0, E2 0, E3 0, E4 0}
LIN {X 588.866, Y 334.557, Z 415.888, A -110.612, B 84.801, C -94.37, E1 0, E2 0, E3 0, E4 0}
LIN {X 587.622, Y 329.733, Z 416.338, A -110.612, B 84.801, C -94.37, E1 0, E2 0, E3 0, E4 0}
LIN {X 511.579, Y 351.912, Z 416.885, A -110.612, B 84.801, C -94.37, E1 0, E2 0, E3 0, E4 0}
LIN {X 510.509, Y 347.037, Z 417.335, A -110.612, B 84.801, C -94.37, E1 0, E2 0, E3 0, E4 0}
LIN {X 567.244, Y 330.489, Z 416.927, A -110.612, B 84.801, C -94.37, E1 0, E2 0, E3 0, E4 0}
LIN {X 546.745, Y 331.281, Z 417.516, A -110.612, B 84.801, C -94.37, E1 0, E2 0, E3 0, E4 0}
LIN {X 509.072, Y 342.269, Z 417.787, A -110.612, B 84.801, C -94.37, E1 0, E2 0, E3 0, E4 0}
LIN {X 507.766, Y 337.463, Z 418.238, A -110.612, B 84.801, C -94.37, E1 0, E2 0, E3 0, E4 0}
LIN {X 528.693, Y 331.359, Z 418.087, A -110.612, B 84.801, C -94.37, E1 0, E2 0, E3 0, E4 0}
LIN {X 510.536, Y 331.468, Z 418.66, A -110.612, B 84.801, C -94.37, E1 0, E2 0, E3 0, E4 0}
LIN {X 506.421, Y 332.668, Z 418.689, A -110.612, B 84.801, C -94.37, E1 0, E2 0, E3 0, E4 0}
LIN {X 595.87, Y 358.45, Z 413.628, A -110.612, B 84.801, C -94.37, E1 0, E2 0, E3 0, E4 0}
LIN {X 595.801, Y 358.265, Z 411.463, A -110.612, B 84.801, C -94.37, E1 0, E2 0, E3 0, E4 0}
LIN {X 594.691, Y 358.589, Z 411.471, A -110.612, B 84.801, C -94.37, E1 0, E2 0, E3 0, E4 0}
LIN {X 553.839, Y 365.317, Z 412.207, A -110.612, B 84.801, C -94.37, E1 0, E2 0, E3 0, E4 0}
LIN {X 595.986, Y 353.024, Z 411.904, A -110.612, B 84.801, C -94.37, E1 0, E2 0, E3 0, E4 0}
LIN {X 549.15, Y 366.684, Z 412.241, A -110.612, B 84.801, C -94.37, E1 0, E2 0, E3 0, E4 0}
LIN {X 545.197, Y 367.837, Z 412.269, A -110.612, B 84.801, C -94.37, E1 0, E2 0, E3 0, E4 0}
LIN {X 516.002, Y 371.165, Z 412.921, A -110.612, B 84.801, C -94.37, E1 0, E2 0, E3 0, E4 0}
LIN {X 594.856, Y 348.167, Z 412.354, A -110.612, B 84.801, C -94.37, E1 0, E2 0, E3 0, E4 0}
LIN {X 592.931, Y 343.541, Z 412.81, A -110.612, B 84.801, C -94.37, E1 0, E2 0, E3 0, E4 0}
LIN {X 514.622, Y 366.381, Z 413.373, A -110.612, B 84.801, C -94.37, E1 0, E2 0, E3 0, E4 0}
LIN {X 513.49, Y 361.524, Z 413.822, A -110.612, B 84.801, C -94.37, E1 0, E2 0, E3 0, E4 0}
LIN {X 591.509, Y 338.769, Z 413.261, A -110.612, B 84.801, C -94.37, E1 0, E2 0, E3 0, E4 0}
LIN {X 590.259, Y 333.946, Z 413.712, A -110.612, B 84.801, C -94.37, E1 0, E2 0, E3 0, E4 0}
LIN {X 512.104, Y 356.741, Z 414.274, A -110.612, B 84.801, C -94.37, E1 0, E2 0, E3 0, E4 0}
LIN {X 510.988, Y 351.88, Z 414.724, A -110.612, B 84.801, C -94.37, E1 0, E2 0, E3 0, E4 0}
LIN {X 588.624, Y 329.236, Z 414.165, A -110.612, B 84.801, C -94.37, E1 0, E2 0, E3 0, E4 0}
LIN {X 567.265, Y 330.279, Z 414.761, A -110.612, B 84.801, C -94.37, E1 0, E2 0, E3 0, E4 0}
LIN {X 509.789, Y 347.042, Z 415.174, A -110.612, B 84.801, C -94.37, E1 0, E2 0, E3 0, E4 0}
LIN {X 508.271, Y 342.298, Z 415.627, A -110.612, B 84.801, C -94.37, E1 0, E2 0, E3 0, E4 0}
LIN {X 546.753, Y 331.074, Z 415.35, A -110.612, B 84.801, C -94.37, E1 0, E2 0, E3 0, E4 0}
LIN {X 528.68, Y 331.158, Z 415.922, A -110.612, B 84.801, C -94.37, E1 0, E2 0, E3 0, E4 0}
LIN {X 507.076, Y 337.459, Z 416.077, A -110.612, B 84.801, C -94.37, E1 0, E2 0, E3 0, E4 0}
LIN {X 505.576, Y 332.71, Z 416.53, A -110.612, B 84.801, C -94.37, E1 0, E2 0, E3 0, E4 0}
LIN {X 510.576, Y 331.251, Z 416.494, A -110.612, B 84.801, C -94.37, E1 0, E2 0, E3 0, E4 0}
LIN {X 597.583, Y 357.745, Z 411.451, A -110.612, B 84.801, C -94.37, E1 0, E2 0, E3 0, E4 0}
LIN {X 597.513, Y 357.561, Z 409.286, A -110.612, B 84.801, C -94.37, E1 0, E2 0, E3 0, E4 0}
LIN {X 596.245, Y 357.931, Z 409.295, A -110.612, B 84.801, C -94.37, E1 0, E2 0, E3 0, E4 0}
LIN {X 544.85, Y 367.734, Z 410.107, A -110.612, B 84.801, C -94.37, E1 0, E2 0, E3 0, E4 0}
LIN {X 597.237, Y 352.455, Z 409.73, A -110.612, B 84.801, C -94.37, E1 0, E2 0, E3 0, E4 0}
LIN {X 544.643, Y 367.794, Z 410.108, A -110.612, B 84.801, C -94.37, E1 0, E2 0, E3 0, E4 0}
LIN {X 543.702, Y 368.069, Z 410.115, A -110.612, B 84.801, C -94.37, E1 0, E2 0, E3 0, E4 0}
LIN {X 515.301, Y 371.165, Z 410.761, A -110.612, B 84.801, C -94.37, E1 0, E2 0, E3 0, E4 0}
LIN {X 595.916, Y 347.653, Z 410.181, A -110.612, B 84.801, C -94.37, E1 0, E2 0, E3 0, E4 0}
LIN {X 594.161, Y 342.978, Z 410.635, A -110.612, B 84.801, C -94.37, E1 0, E2 0, E3 0, E4 0}
LIN {X 513.516, Y 366.499, Z 411.215, A -110.612, B 84.801, C -94.37, E1 0, E2 0, E3 0, E4 0}
LIN {X 512.298, Y 361.667, Z 411.666, A -110.612, B 84.801, C -94.37, E1 0, E2 0, E3 0, E4 0}
LIN {X 592.832, Y 338.178, Z 411.087, A -110.612, B 84.801, C -94.37, E1 0, E2 0, E3 0, E4 0}
LIN {X 591.46, Y 333.392, Z 411.538, A -110.612, B 84.801, C -94.37, E1 0, E2 0, E3 0, E4 0}
LIN {X 511.321, Y 356.765, Z 412.114, A -110.612, B 84.801, C -94.37, E1 0, E2 0, E3 0, E4 0}
LIN {X 510.194, Y 351.906, Z 412.564, A -110.612, B 84.801, C -94.37, E1 0, E2 0, E3 0, E4 0}
LIN {X 589.426, Y 328.798, Z 411.995, A -110.612, B 84.801, C -94.37, E1 0, E2 0, E3 0, E4 0}
LIN {X 567.25, Y 330.078, Z 412.596, A -110.612, B 84.801, C -94.37, E1 0, E2 0, E3 0, E4 0}
LIN {X 509.203, Y 347.009, Z 413.013, A -110.612, B 84.801, C -94.37, E1 0, E2 0, E3 0, E4 0}
LIN {X 507.762, Y 342.242, Z 413.465, A -110.612, B 84.801, C -94.37, E1 0, E2 0, E3 0, E4 0}
LIN {X 546.713, Y 330.881, Z 413.185, A -110.612, B 84.801, C -94.37, E1 0, E2 0, E3 0, E4 0}
LIN {X 528.626, Y 330.97, Z 413.757, A -110.612, B 84.801, C -94.37, E1 0, E2 0, E3 0, E4 0}
LIN {X 506.343, Y 337.469, Z 413.917, A -110.612, B 84.801, C -94.37, E1 0, E2 0, E3 0, E4 0}
LIN {X 504.978, Y 332.68, Z 414.369, A -110.612, B 84.801, C -94.37, E1 0, E2 0, E3 0, E4 0}
LIN {X 510.559, Y 331.052, Z 414.328, A -110.612, B 84.801, C -94.37, E1 0, E2 0, E3 0, E4 0}
LIN {X 593.131, Y 358.839, Z 409.317, A -110.612, B 84.801, C -94.37, E1 0, E2 0, E3 0, E4 0}
LIN {X 593.062, Y 358.655, Z 407.152, A -110.612, B 84.801, C -94.37, E1 0, E2 0, E3 0, E4 0}
LIN {X 598.744, Y 356.998, Z 407.111, A -110.612, B 84.801, C -94.37, E1 0, E2 0, E3 0, E4 0}
LIN {X 598.302, Y 351.939, Z 407.556, A -110.612, B 84.801, C -94.37, E1 0, E2 0, E3 0, E4 0}
LIN {X 543.828, Y 367.827, Z 407.948, A -110.612, B 84.801, C -94.37, E1 0, E2 0, E3 0, E4 0}
LIN {X 514.778, Y 371.113, Z 408.599, A -110.612, B 84.801, C -94.37, E1 0, E2 0, E3 0, E4 0}
LIN {X 596.757, Y 347.203, Z 408.009, A -110.612, B 84.801, C -94.37, E1 0, E2 0, E3 0, E4 0}
LIN {X 595.319, Y 342.436, Z 408.461, A -110.612, B 84.801, C -94.37, E1 0, E2 0, E3 0, E4 0}
LIN {X 512.939, Y 366.463, Z 409.054, A -110.612, B 84.801, C -94.37, E1 0, E2 0, E3 0, E4 0}
LIN {X 511.685, Y 361.641, Z 409.505, A -110.612, B 84.801, C -94.37, E1 0, E2 0, E3 0, E4 0}
LIN {X 594.1, Y 337.604, Z 408.912, A -110.612, B 84.801, C -94.37, E1 0, E2 0, E3 0, E4 0}
LIN {X 592.623, Y 332.848, Z 409.364, A -110.612, B 84.801, C -94.37, E1 0, E2 0, E3 0, E4 0}
LIN {X 510.581, Y 356.776, Z 409.954, A -110.612, B 84.801, C -94.37, E1 0, E2 0, E3 0, E4 0}
LIN {X 509.482, Y 351.91, Z 410.404, A -110.612, B 84.801, C -94.37, E1 0, E2 0, E3 0, E4 0}
LIN {X 589.429, Y 328.592, Z 409.829, A -110.612, B 84.801, C -94.37, E1 0, E2 0, E3 0, E4 0}
LIN {X 567.291, Y 329.862, Z 410.43, A -110.612, B 84.801, C -94.37, E1 0, E2 0, E3 0, E4 0}
LIN {X 508.549, Y 346.995, Z 410.852, A -110.612, B 84.801, C -94.37, E1 0, E2 0, E3 0, E4 0}
LIN {X 507.22, Y 342.195, Z 411.304, A -110.612, B 84.801, C -94.37, E1 0, E2 0, E3 0, E4 0}
LIN {X 546.72, Y 330.675, Z 411.019, A -110.612, B 84.801, C -94.37, E1 0, E2 0, E3 0, E4 0}
LIN {X 528.612, Y 330.769, Z 411.591, A -110.612, B 84.801, C -94.37, E1 0, E2 0, E3 0, E4 0}
LIN {X 505.868, Y 337.402, Z 411.755, A -110.612, B 84.801, C -94.37, E1 0, E2 0, E3 0, E4 0}
LIN {X 504.405, Y 332.642, Z 412.207, A -110.612, B 84.801, C -94.37, E1 0, E2 0, E3 0, E4 0}
LIN {X 510.597, Y 330.836, Z 412.163, A -110.612, B 84.801, C -94.37, E1 0, E2 0, E3 0, E4 0}
LIN {X 589.776, Y 359.613, Z 407.176, A -110.612, B 84.801, C -94.37, E1 0, E2 0, E3 0, E4 0}
LIN {X 589.706, Y 359.429, Z 405.011, A -110.612, B 84.801, C -94.37, E1 0, E2 0, E3 0, E4 0}
LIN {X 599.364, Y 356.612, Z 404.942, A -110.612, B 84.801, C -94.37, E1 0, E2 0, E3 0, E4 0}
LIN {X 599.159, Y 351.485, Z 405.385, A -110.612, B 84.801, C -94.37, E1 0, E2 0, E3 0, E4 0}
LIN {X 540.024, Y 368.732, Z 405.81, A -110.612, B 84.801, C -94.37, E1 0, E2 0, E3 0, E4 0}
LIN {X 514.381, Y 371.024, Z 406.436, A -110.612, B 84.801, C -94.37, E1 0, E2 0, E3 0, E4 0}
LIN {X 597.957, Y 346.649, Z 405.835, A -110.612, B 84.801, C -94.37, E1 0, E2 0, E3 0, E4 0}
LIN {X 596.463, Y 341.897, Z 406.288, A -110.612, B 84.801, C -94.37, E1 0, E2 0, E3 0, E4 0}
LIN {X 512.653, Y 366.341, Z 406.89, A -110.612, B 84.801, C -94.37, E1 0, E2 0, E3 0, E4 0}
LIN {X 511.122, Y 361.601, Z 407.343, A -110.612, B 84.801, C -94.37, E1 0, E2 0, E3 0, E4 0}
LIN {X 595.192, Y 337.081, Z 406.739, A -110.612, B 84.801, C -94.37, E1 0, E2 0, E3 0, E4 0}
LIN {X 593.592, Y 332.36, Z 407.192, A -110.612, B 84.801, C -94.37, E1 0, E2 0, E3 0, E4 0}
LIN {X 510.103, Y 356.711, Z 407.792, A -110.612, B 84.801, C -94.37, E1 0, E2 0, E3 0, E4 0}
LIN {X 509.017, Y 351.841, Z 408.242, A -110.612, B 84.801, C -94.37, E1 0, E2 0, E3 0, E4 0}
LIN {X 589.381, Y 328.402, Z 407.664, A -110.612, B 84.801, C -94.37, E1 0, E2 0, E3 0, E4 0}
LIN {X 567.262, Y 329.666, Z 408.264, A -110.612, B 84.801, C -94.37, E1 0, E2 0, E3 0, E4 0}
LIN {X 508.08, Y 346.927, Z 408.69, A -110.612, B 84.801, C -94.37, E1 0, E2 0, E3 0, E4 0}
LIN {X 506.821, Y 342.107, Z 409.141, A -110.612, B 84.801, C -94.37, E1 0, E2 0, E3 0, E4 0}
LIN {X 546.673, Y 330.484, Z 408.854, A -110.612, B 84.801, C -94.37, E1 0, E2 0, E3 0, E4 0}
LIN {X 528.555, Y 330.581, Z 409.426, A -110.612, B 84.801, C -94.37, E1 0, E2 0, E3 0, E4 0}
LIN {X 505.52, Y 337.299, Z 409.592, A -110.612, B 84.801, C -94.37, E1 0, E2 0, E3 0, E4 0}
LIN {X 504.056, Y 332.539, Z 410.044, A -110.612, B 84.801, C -94.37, E1 0, E2 0, E3 0, E4 0}
LIN {X 510.566, Y 330.641, Z 409.997, A -110.612, B 84.801, C -94.37, E1 0, E2 0, E3 0, E4 0}
LIN {X 587.709, Y 360.012, Z 405.026, A -110.612, B 84.801, C -94.37, E1 0, E2 0, E3 0, E4 0}
LIN {X 587.64, Y 359.827, Z 402.861, A -110.612, B 84.801, C -94.37, E1 0, E2 0, E3 0, E4 0}
LIN {X 599.598, Y 356.339, Z 402.775, A -110.612, B 84.801, C -94.37, E1 0, E2 0, E3 0, E4 0}
LIN {X 599.248, Y 351.255, Z 403.219, A -110.612, B 84.801, C -94.37, E1 0, E2 0, E3 0, E4 0}
LIN {X 539.695, Y 368.624, Z 403.647, A -110.612, B 84.801, C -94.37, E1 0, E2 0, E3 0, E4 0}
LIN {X 514.179, Y 370.879, Z 404.272, A -110.612, B 84.801, C -94.37, E1 0, E2 0, E3 0, E4 0}
LIN {X 598.141, Y 346.39, Z 403.668, A -110.612, B 84.801, C -94.37, E1 0, E2 0, E3 0, E4 0}
LIN {X 596.981, Y 341.542, Z 404.119, A -110.612, B 84.801, C -94.37, E1 0, E2 0, E3 0, E4 0}
LIN {X 512.315, Y 366.235, Z 404.727, A -110.612, B 84.801, C -94.37, E1 0, E2 0, E3 0, E4 0}
LIN {X 510.918, Y 361.456, Z 405.179, A -110.612, B 84.801, C -94.37, E1 0, E2 0, E3 0, E4 0}
LIN {X 595.625, Y 336.75, Z 404.57, A -110.612, B 84.801, C -94.37, E1 0, E2 0, E3 0, E4 0}
LIN {X 594.478, Y 331.898, Z 405.02, A -110.612, B 84.801, C -94.37, E1 0, E2 0, E3 0, E4 0}
LIN {X 509.793, Y 356.597, Z 405.629, A -110.612, B 84.801, C -94.37, E1 0, E2 0, E3 0, E4 0}
LIN {X 508.839, Y 351.688, Z 406.077, A -110.612, B 84.801, C -94.37, E1 0, E2 0, E3 0, E4 0}
LIN {X 589.357, Y 328.204, Z 405.499, A -110.612, B 84.801, C -94.37, E1 0, E2 0, E3 0, E4 0}
LIN {X 567.266, Y 329.46, Z 406.099, A -110.612, B 84.801, C -94.37, E1 0, E2 0, E3 0, E4 0}
LIN {X 507.926, Y 346.767, Z 406.526, A -110.612, B 84.801, C -94.37, E1 0, E2 0, E3 0, E4 0}
LIN {X 506.658, Y 341.95, Z 406.977, A -110.612, B 84.801, C -94.37, E1 0, E2 0, E3 0, E4 0}
LIN {X 546.652, Y 330.285, Z 406.689, A -110.612, B 84.801, C -94.37, E1 0, E2 0, E3 0, E4 0}
LIN {X 528.518, Y 330.387, Z 407.261, A -110.612, B 84.801, C -94.37, E1 0, E2 0, E3 0, E4 0}
LIN {X 505.372, Y 337.138, Z 407.428, A -110.612, B 84.801, C -94.37, E1 0, E2 0, E3 0, E4 0}
LIN {X 504.102, Y 332.321, Z 407.878, A -110.612, B 84.801, C -94.37, E1 0, E2 0, E3 0, E4 0}
LIN {X 510.568, Y 330.436, Z 407.832, A -110.612, B 84.801, C -94.37, E1 0, E2 0, E3 0, E4 0}
LIN {X 587.397, Y 359.898, Z 402.862, A -110.612, B 84.801, C -94.37, E1 0, E2 0, E3 0, E4 0}
LIN {X 587.328, Y 359.713, Z 400.697, A -110.612, B 84.801, C -94.37, E1 0, E2 0, E3 0, E4 0}
LIN {X 599.563, Y 356.145, Z 400.609, A -110.612, B 84.801, C -94.37, E1 0, E2 0, E3 0, E4 0}
LIN {X 599.29, Y 351.038, Z 401.053, A -110.612, B 84.801, C -94.37, E1 0, E2 0, E3 0, E4 0}
LIN {X 538.471, Y 368.776, Z 401.491, A -110.612, B 84.801, C -94.37, E1 0, E2 0, E3 0, E4 0}
LIN {X 514.261, Y 370.65, Z 402.106, A -110.612, B 84.801, C -94.37, E1 0, E2 0, E3 0, E4 0}
LIN {X 598.284, Y 346.144, Z 401.502, A -110.612, B 84.801, C -94.37, E1 0, E2 0, E3 0, E4 0}
LIN {X 597.105, Y 341.301, Z 401.952, A -110.612, B 84.801, C -94.37, E1 0, E2 0, E3 0, E4 0}
LIN {X 512.526, Y 365.969, Z 402.561, A -110.612, B 84.801, C -94.37, E1 0, E2 0, E3 0, E4 0}
LIN {X 510.836, Y 361.275, Z 403.015, A -110.612, B 84.801, C -94.37, E1 0, E2 0, E3 0, E4 0}
LIN {X 596.065, Y 336.417, Z 402.401, A -110.612, B 84.801, C -94.37, E1 0, E2 0, E3 0, E4 0}
LIN {X 595.071, Y 331.52, Z 402.85, A -110.612, B 84.801, C -94.37, E1 0, E2 0, E3 0, E4 0}
LIN {X 509.821, Y 356.384, Z 403.464, A -110.612, B 84.801, C -94.37, E1 0, E2 0, E3 0, E4 0}
LIN {X 508.846, Y 351.481, Z 403.912, A -110.612, B 84.801, C -94.37, E1 0, E2 0, E3 0, E4 0}
LIN {X 589.301, Y 328.016, Z 403.333, A -110.612, B 84.801, C -94.37, E1 0, E2 0, E3 0, E4 0}
LIN {X 567.227, Y 329.267, Z 403.934, A -110.612, B 84.801, C -94.37, E1 0, E2 0, E3 0, E4 0}
LIN {X 507.881, Y 346.576, Z 404.361, A -110.612, B 84.801, C -94.37, E1 0, E2 0, E3 0, E4 0}
LIN {X 506.891, Y 341.678, Z 404.81, A -110.612, B 84.801, C -94.37, E1 0, E2 0, E3 0, E4 0}
LIN {X 546.597, Y 330.097, Z 404.524, A -110.612, B 84.801, C -94.37, E1 0, E2 0, E3 0, E4 0}
LIN {X 528.454, Y 330.201, Z 405.096, A -110.612, B 84.801, C -94.37, E1 0, E2 0, E3 0, E4 0}
LIN {X 505.6, Y 336.867, Z 405.261, A -110.612, B 84.801, C -94.37, E1 0, E2 0, E3 0, E4 0}
LIN {X 504.543, Y 331.988, Z 405.71, A -110.612, B 84.801, C -94.37, E1 0, E2 0, E3 0, E4 0}
LIN {X 510.528, Y 330.243, Z 405.667, A -110.612, B 84.801, C -94.37, E1 0, E2 0, E3 0, E4 0}
LIN {X 586.77, Y 359.876, Z 400.702, A -110.612, B 84.801, C -94.37, E1 0, E2 0, E3 0, E4 0}
LIN {X 586.701, Y 359.692, Z 398.537, A -110.612, B 84.801, C -94.37, E1 0, E2 0, E3 0, E4 0}
LIN {X 599.52, Y 355.953, Z 398.444, A -110.612, B 84.801, C -94.37, E1 0, E2 0, E3 0, E4 0}
LIN {X 599.228, Y 350.851, Z 398.888, A -110.612, B 84.801, C -94.37, E1 0, E2 0, E3 0, E4 0}
LIN {X 535.28, Y 369.502, Z 399.348, A -110.612, B 84.801, C -94.37, E1 0, E2 0, E3 0, E4 0}
LIN {X 514.935, Y 370.249, Z 399.936, A -110.612, B 84.801, C -94.37, E1 0, E2 0, E3 0, E4 0}
LIN {X 598.27, Y 345.944, Z 399.337, A -110.612, B 84.801, C -94.37, E1 0, E2 0, E3 0, E4 0}
LIN {X 596.982, Y 341.132, Z 399.788, A -110.612, B 84.801, C -94.37, E1 0, E2 0, E3 0, E4 0}
LIN {X 512.784, Y 365.689, Z 400.393, A -110.612, B 84.801, C -94.37, E1 0, E2 0, E3 0, E4 0}
LIN {X 511.353, Y 360.919, Z 400.845, A -110.612, B 84.801, C -94.37, E1 0, E2 0, E3 0, E4 0}
LIN {X 596.095, Y 336.204, Z 400.236, A -110.612, B 84.801, C -94.37, E1 0, E2 0, E3 0, E4 0}
LIN {X 595.03, Y 331.327, Z 400.685, A -110.612, B 84.801, C -94.37, E1 0, E2 0, E3 0, E4 0}
LIN {X 510.172, Y 356.077, Z 401.296, A -110.612, B 84.801, C -94.37, E1 0, E2 0, E3 0, E4 0}
LIN {X 509.351, Y 351.129, Z 401.743, A -110.612, B 84.801, C -94.37, E1 0, E2 0, E3 0, E4 0}
LIN {X 589.212, Y 327.837, Z 401.169, A -110.612, B 84.801, C -94.37, E1 0, E2 0, E3 0, E4 0}
LIN {X 567.227, Y 329.062, Z 401.769, A -110.612, B 84.801, C -94.37, E1 0, E2 0, E3 0, E4 0}
LIN {X 508.301, Y 346.249, Z 402.192, A -110.612, B 84.801, C -94.37, E1 0, E2 0, E3 0, E4 0}
LIN {X 507.267, Y 341.363, Z 402.642, A -110.612, B 84.801, C -94.37, E1 0, E2 0, E3 0, E4 0}
LIN {X 546.596, Y 329.892, Z 402.359, A -110.612, B 84.801, C -94.37, E1 0, E2 0, E3 0, E4 0}
LIN {X 528.42, Y 330.007, Z 402.931, A -110.612, B 84.801, C -94.37, E1 0, E2 0, E3 0, E4 0}
LIN {X 506.184, Y 336.492, Z 403.091, A -110.612, B 84.801, C -94.37, E1 0, E2 0, E3 0, E4 0}
LIN {X 505.029, Y 331.642, Z 403.541, A -110.612, B 84.801, C -94.37, E1 0, E2 0, E3 0, E4 0}
LIN {X 510.534, Y 330.036, Z 403.502, A -110.612, B 84.801, C -94.37, E1 0, E2 0, E3 0, E4 0}
PTP {X 556.311, Y 346.712, Z 474.273, A -110.612, B 84.801, C -94.37, E1 0, E2 0, E3 0, E4 0, S 'B010'}
PTP {A1 5, A2 -90, A3 100, A4 5, A5 -10, A6 -5, E1 0, E2 0, E3 0, E4 0} C_PTP

END
